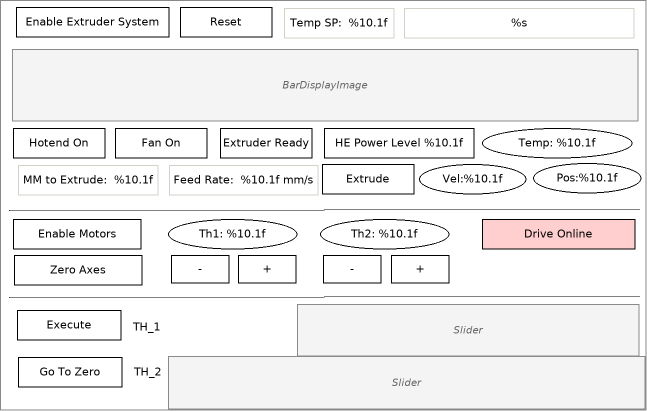
VISUALIZATION Visualization  // 647x411
    RoundedRectangle (16,7 153x30), "Enable Extruder System", colour toggle: GVL_AxisCtrl.bExtruderSystemEnable
        toggle GVL_AxisCtrl.bExtruderSystemEnable
    RoundedRectangle (13,128 92x30), "Hotend On", colour toggle: GVL_IO.bEnableHotend
    RoundedRectangle (115,128 92x30), "Fan On", colour toggle: GVL_IO.bFan
    BarDisplayImage (12,49 626x72), value: GVL_IO.lrHotendTemp, invisible if: FALSE, style: BarDisplayImage-Gray, scale format: %.1f, scale 0..300
    RoundedRectangle (180,7 92x30), "Reset"
        tap GVL_AxisCtrl.bExtruderSystemReset
        OnMouseDown: execute { GVL_AxisCtrl.bExtruderSystemEnable := FALSE; }
    Ellipse (482,128 150x30), "Temp: %10.1f", text variable: GVL_IO.lrHotendTemp
    RoundedRectangle (324,128 150x30), "HE Power Level %10.1f", text variable: GVL_IO.iHotendPowerLevel
    Textfield (284,8 110x30), "Temp SP: %10.1f", text variable: GVL_AxisCtrl.lrHotEndTempSP
        OnMouseDown: write GVL_AxisCtrl.lrHotEndTempSP via InputWithLimits, min 180, max 240
    RoundedRectangle (220,128 92x30), "Extruder Ready", colour toggle: GVL_AxisCtrl.bExtruderReady
    RoundedRectangle (322,164 92x30), "Extrude", input disabled if: NOT GVL_AxisCtrl.bExtruderReady
        tap GVL_AxisCtrl.bExtruder_AxisMoveHMI
    Textfield (404,8 230x30), "%s", text variable: GVL_AxisCtrl.sExtruderSystemStatus
    Textfield (18,165 140x30), "MM to Extrude: %10.1f", text variable: GVL_AxisCtrl.lrExtruder_AxisTarget
        OnMouseDown: write GVL_AxisCtrl.lrExtruder_AxisTarget via InputWithLimits, min 0, max 1000
    Textfield (169,165 149x30), "Feed Rate: %10.1f mm/s", text variable: GVL_AxisCtrl.lrExtruder_AxisVelocity
        OnMouseDown: write GVL_AxisCtrl.lrExtruder_AxisVelocity via InputWithLimits, min 0, max 4
    Ellipse (533,163 108x30), "Pos:%10.1f", text variable: GVL_NC.Extruder_AXIS.NcToPlc.ActPos
    Ellipse (419,164 107x30), "Vel:%10.1f", text variable: GVL_NC.Extruder_AXIS.NcToPlc.ActVelo
    Line (9,210) (639,209)
    RoundedRectangle (13,219 128x30), "Enable Motors", colour toggle: GVL_AxisCtrl.bEnableGimbal
        toggle GVL_AxisCtrl.bEnableGimbal
    RoundedRectangle (482,219 153x30), "Drive Online", colour toggle: GVL_AxisCtrl.bAllAxisEnabled
    RoundedRectangle (14,255 128x30), "Zero Axes"
        tap GVL_AxisCtrl.bZeroAxes
        OnMouseDown: execute {  }
    Ellipse (168,219 129x30), "Th1: %10.1f", text variable: GVL_NC.Th1_AXIS.NcToPlc.ActPos
    Ellipse (320,219 129x30), "Th2: %10.1f", text variable: GVL_NC.Th2_AXIS.NcToPlc.ActPos
    RoundedRectangle (171,255 58x28), "-"
        tap GVL_AxisCtrl.bJogTh1_Neg
    RoundedRectangle (391,255 58x28), "+"
        tap GVL_AxisCtrl.bJogTh2_Pos
    RoundedRectangle (238,255 58x28), "+"
        tap GVL_AxisCtrl.bJogTh1_Pos p3779583253=TRUE
    RoundedRectangle (323,255 58x28), "-"
        tap GVL_AxisCtrl.bJogTh2_Neg
    Line (9,297) (639,296)
    Slider (297,304 342x52), variable: GVL_AxisCtrl.lrTh1Target, scale -16..35
    Slider (168,356 477x53), variable: GVL_AxisCtrl.lrTh2Target, scale -160..160
    Label (122,312 50x30), "TH_1"
    RoundedRectangle (18,357 104x30), "Go To Zero"
        OnMouseDown: execute { GVL_AxisCtrl.lrTh1Target := 0; GVL_AxisCtrl.lrTh2Target := 0; GVL_AxisCtrl.bExecuteMove := TRUE; }
    Label (107,357 82x30), "TH_2"
    RoundedRectangle (17,310 104x30), "Execute"
        tap GVL_AxisCtrl.bExecuteMove
        OnMouseDown: execute {  }
END_VISUALIZATION

(* stored: Version 1.1.0.1, ProductVersion 3.1.4024.2
   Visu Visualization: Id {57b130c3-747d-42f7-870c-37d094ed37fa} *)
